(* Logix 5000 project; controller KTC_lab5_tank vendor 1 type 14 code 149 rev 30.11; software revision 30.00 *)

TASK MainTask (continuous, watchdog 500 ms) : MainProgram

MODULES
   Local : vendor 1 type 14 code 149 (Compact 0, rev 30.11)
      Discrete_IO : Embedded (Compact 1, rev 3.1, Output RPI 20 ms)
END_MODULES

PROGRAM MainProgram   (* main routine MainRoutine *)
VAR
   pl1 : ALIAS FOR Local:1:O.Data.0;   // inlet valve
   pl2 : ALIAS FOR Local:1:O.Data;   // outlet valve
   pl3 : ALIAS FOR Local:1:O.Data.3;   // water heat
   pos1 : ALIAS FOR Local:1:I.Data.3;   // max water level
   pos2 : ALIAS FOR Local:1:O.Data.2;   // outlet valve
   pos3 : ALIAS FOR Local:1:I.Data.0;   // low water
   pos4 : ALIAS FOR Local:1:I.Data.5;   // high temp
   pos5 : ALIAS FOR Local:1:I.Data.4;   // low temp
   pos6 : ALIAS FOR Local:1:O.Data.3;   // heat
END_VAR

ROUTINE MainRoutine   (* ladder *)
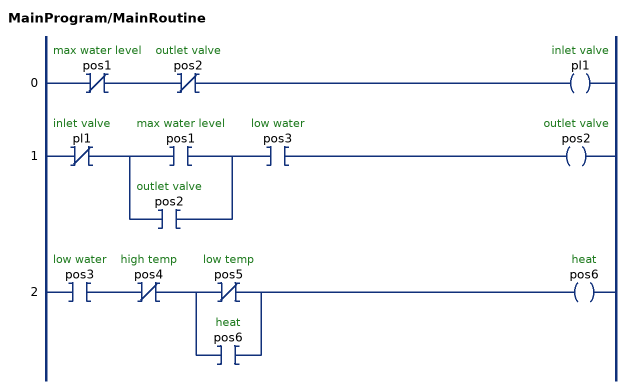
   0: XIO(pos1)XIO(pos2)OTE(pl1);
   1: XIO(pl1)[XIC(pos1) ,XIC(pos2) ]XIC(pos3)OTE(pos2);
   2: XIC(pos3)XIO(pos4)[XIO(pos5) ,XIC(pos6) ]OTE(pos6);
END_ROUTINE
END_PROGRAM
